TYPE TcoTixonGenericControl : 
STRUCT	
	

	
	{attribute addProperty Name "<#Feeding A #> - q1"}
	FeedingA: BOOL;
	{attribute addProperty Name "<#Separe component#> - q2"}
	SepareComponent : BOOL;
	{attribute addProperty Name "<#Blow A#> - q3"}
	BlowAValve  : BOOL;
	{attribute addProperty Name "<#Red led#> - q4"}
	RedLed : BOOL;
	{attribute addProperty Name "<#Green led#> - q5"}
	GreenLed  : BOOL;
	{attribute addProperty Name "<#Hooper#> - q6"}
	Hooper  : BOOL;

	
END_STRUCT
END_TYPE

(* stored: Version 1.1.0.1, ProductVersion 3.1.4024.12
   DUT TcoTixonGenericControl: Id {793867f9-8255-082a-1b3c-92fbb08ea703} *)
